{attribute 'qualified_only'}
VAR_GLOBAL
	Axis1		:AXIS_REF;
	fbAxis		:FB_Axis;
	
	bPowrOn		:BOOL;
	
//----------------------HMI-----------------
	hmiPowerOn	:BOOL;
	hmiStop		:BOOL;
	hmiMoveVelo		:BOOL;
	hmiHome			:BOOL;
	hmiDummyHomeSensor		:BOOL;
	hmiSetPosition			:BOOL;
	hmiMoveRelative			:BOOL;
	hmiLActPos				:LREAL;
	hmiJogFor				:BOOL;
	hmiJogBack				:BOOL;
	hmiManualJog			:BOOL;
//-----------------------HMI-----------------

//-----------------Log---------------------
	fbLocalTime: FB_LocalSystemTime := (bEnable:= TRUE, dwCycle:= 1);
	DateTimeNow		:STRING;
	//LogBufferArray: ARRAY[1..10] OF STRING := ['a','b','c','d','e','f','g','7','9','10'];
	LogBufferArray: ARRAY[1..10] OF STRING;
	LogBufferIndex	:INT;
	sFilePath		:STRING :='C:\TempSample\';
	

//-----------------Log---------------------

	
	
END_VAR

(* stored: Version 1.1.0.1, ProductVersion 3.1.4022.16
   GVL GVL_General: Id {87d87095-3528-4336-963a-cc20e50b28e6} *)
